FUNCTION_BLOCK Faults4
VAR_INPUT
END_VAR
VAR_OUTPUT
END_VAR
VAR
END_VAR

END_FUNCTION_BLOCK

(* stored: Version 1.1.0.1, ProductVersion 3.1.4024.11
   POU Faults4: Id {5e3e73bf-0b44-43c7-93a4-c3cd3f239304}, SpecialFunc None *)
